SYSTEM FbeTestProject
  (* Standard: Test standard; Classification: Test; ApplicationDomain: GASR; Function: For testing; Type: Test; Description: System created for test purposes only *)
  (* Version 1.0, 2024-08-05, cabral, GASR-UDESC, None *)
  APPLICATION MainApp
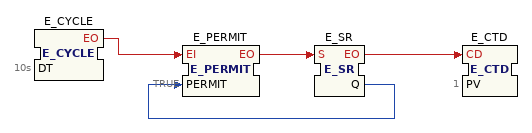
    FBS
      E_SR : E_SR; (* Event-driven bistable *)
      E_PERMIT : E_PERMIT(PERMIT := TRUE); (* permissive propagation of an event *)
      E_CYCLE : E_CYCLE(DT := 10s); (* Peroidic event generator *)
      E_CTD : E_CTD(PV := 1); (* Event-Driven Down Counter *)
    END_FBS
    EVENT_CONNECTIONS
      E_CYCLE.EO TO E_PERMIT.EI;
      E_PERMIT.EO TO E_SR.S;
      E_SR.EO TO E_CTD.CD;
    END_CONNECTIONS
    DATA_CONNECTIONS
      E_SR.Q TO E_PERMIT.PERMIT;
    END_CONNECTIONS
  END_APPLICATION
  APPLICATION SumApp
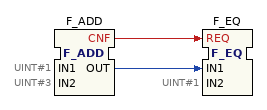
    FBS
      F_ADD : F_ADD(IN1 := UINT#1, IN2 := UINT#3); (* Adds two number values *)
      F_EQ : F_EQ(IN2 := UINT#1); (* equal *)
    END_FBS
    EVENT_CONNECTIONS
      F_ADD.CNF TO F_EQ.REQ;
    END_CONNECTIONS
    DATA_CONNECTIONS
      F_ADD.OUT TO F_EQ.IN1;
    END_CONNECTIONS
  END_APPLICATION
  APPLICATION MultApp
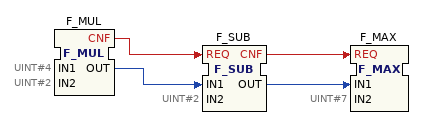
    FBS
      F_MUL : F_MUL(IN1 := UINT#4, IN2 := UINT#2); (* Multiplies two values *)
      F_SUB : F_SUB(IN2 := UINT#2); (* Subtracts two number values *)
      F_MAX : F_MAX(IN2 := UINT#7); (* maximum *)
    END_FBS
    EVENT_CONNECTIONS
      F_MUL.CNF TO F_SUB.REQ;
      F_SUB.CNF TO F_MAX.REQ;
    END_CONNECTIONS
    DATA_CONNECTIONS
      F_MUL.OUT TO F_SUB.IN1;
      F_SUB.OUT TO F_MAX.IN1;
    END_CONNECTIONS
  END_APPLICATION
  DEVICE DEV_FORTE : FORTE_PC
    RESOURCE FST_RES : EMB_RES
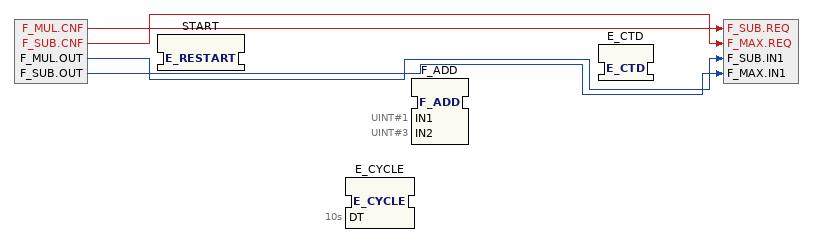
      FBS
        START : E_RESTART; (* Service Interface Function Block Type *)
        F_ADD : F_ADD(IN1 := UINT#1, IN2 := UINT#3); (* Adds two number values *)
        E_CYCLE : E_CYCLE(DT := 10s); (* Peroidic event generator *)
        E_CTD : E_CTD; (* Event-Driven Down Counter *)
      END_FBS
      EVENT_CONNECTIONS
        F_MUL.CNF TO F_SUB.REQ;
        F_SUB.CNF TO F_MAX.REQ;
      END_CONNECTIONS
      DATA_CONNECTIONS
        F_MUL.OUT TO F_SUB.IN1;
        F_SUB.OUT TO F_MAX.IN1;
      END_CONNECTIONS
    END_RESOURCE
    RESOURCE SECOND_RES : EMB_RES
      FBS
        START : E_RESTART; (* Service Interface Function Block Type *)
        E_CTD : E_CTD(PV := 1); (* Event-Driven Down Counter *)
        F_MUL : F_MUL(IN1 := UINT#4, IN2 := UINT#2); (* Multiplies two values *)
      END_FBS
      EVENT_CONNECTIONS
        F_MUL.CNF TO F_SUB.REQ;
        F_SUB.CNF TO F_MAX.REQ;
      END_CONNECTIONS
      DATA_CONNECTIONS
        F_MUL.OUT TO F_SUB.IN1;
        F_SUB.OUT TO F_MAX.IN1;
      END_CONNECTIONS
    END_RESOURCE
    RESOURCE THIRD_RES : EMB_RES
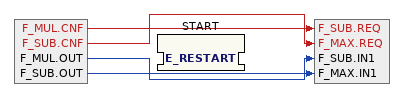
      FBS
        START : E_RESTART; (* Service Interface Function Block Type *)
      END_FBS
      EVENT_CONNECTIONS
        F_MUL.CNF TO F_SUB.REQ;
        F_SUB.CNF TO F_MAX.REQ;
      END_CONNECTIONS
      DATA_CONNECTIONS
        F_MUL.OUT TO F_SUB.IN1;
        F_SUB.OUT TO F_MAX.IN1;
      END_CONNECTIONS
    END_RESOURCE
  END_DEVICE
  DEVICE FORTE : FORTE_PC
    RESOURCE GASR : EMB_RES
      FBS
        START : E_RESTART; (* Service Interface Function Block Type *)
        F_EQ : F_EQ(IN2 := UINT#1); (* equal *)
        FINAL : F_MIN; (* minimum *)
        F_MAX : F_MAX(IN2 := UINT#7); (* maximum *)
      END_FBS
      EVENT_CONNECTIONS
        F_MUL.CNF TO F_SUB.REQ;
        F_SUB.CNF TO F_MAX.REQ;
      END_CONNECTIONS
      DATA_CONNECTIONS
        F_MUL.OUT TO F_SUB.IN1;
        F_SUB.OUT TO F_MAX.IN1;
      END_CONNECTIONS
    END_RESOURCE
  END_DEVICE
  MAPPINGS
    SumApp.F_ADD ON DEV_FORTE.FST_RES.F_ADD;
    SumApp.F_EQ ON FORTE.GASR.F_EQ;
    MainApp.E_CTD ON DEV_FORTE.SECOND_RES.E_CTD;
    MultApp.F_MUL ON DEV_FORTE.SECOND_RES.F_MUL;
    MultApp.F_MAX ON FORTE.GASR.F_MAX;
    MainApp.E_CYCLE ON DEV_FORTE.FST_RES.E_CYCLE;
  END_MAPPINGS
END_SYSTEM
